ABB RobotStudio station: Proyecto_20210527-053903.rsstn

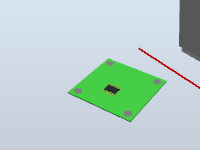
Station Proyecto (saved by RobotStudio 21.1.9443.2)
Controller IRB14000
  mechanical unit ROB_R: IRB14000_0.5_0.5_R, 6 joints, base frame (0, 0, 0) mm
  mechanical unit ROB_R_7: IRB14000_0.5_0.5_R, 1 joints, base frame (0, 0, 0) mm
  mechanical unit ROB_L: IRB14000_0.5_0.5_L, 6 joints, base frame (0, 0, 0) mm
  mechanical unit ROB_L_7: IRB14000_0.5_0.5_L, 1 joints, base frame (0, 0, 0) mm
Layout (positions relative to the parent item):
  - IRB14000_0.5_0.5 [mechanism, from Robots\IRB14000_0.5_0.5__02.rslib] at (0, 0, 0) mm
  - IRB14000_0.5_0.5_R [mechanism, from Robots\IRB14000_0.5_0.5__02.rslib] at (0, 0, 0) mm; joint values [0.0079, -2.3073, -2.3848, 0.4366, 0.2482, 1.2301, -3.4933] (rad or m)
  - IRB14000_0.5_0.5_L [mechanism, from Robots\IRB14000_0.5_0.5__02.rslib] at (0, 0, 0) mm; joint values [-2.0402, -2.3304, 0.9, 0.5715, 0.2248, -0.5734, -1.7213] (rad or m)
  - Part_1 [part] at (100, 0, 0) mm
  - MyTool [mechanism, from Training Objects\myTool.rslib] at (-9.58, -182.61, 198.63) mm, rotated rx -90 ry 76.24 rz -90 deg
  - Chip [part] at (492.85, -76.39, 101.1) mm
  - Drill_holder [mechanism] at (396.94, 21.77, 200.3) mm, rotated rx 106.8 ry 1.53 rz 74.44 deg; joint values [-0.025, 0.0219, 0.0219] (rad or m)
      TCP Tip_holder_mechanism at (-0.08, -53.38, 109.89) mm, rotated rx -73 ry 2 rz -178 deg
      links: L1, L2, L3, L4
  - Part_33 [part]
Attachment: MyTool is attached to IRB14000_0.5_0.5_R / Link7
Attachment: Drill_holder is attached to IRB14000_0.5_0.5_L / Link7
Targets, tools, work objects and paths stored in the station, written as RAPID:
! task T_ROB_R
MODULE CalibData
  PERS tooldata MyTool:=[TRUE,[[31.792631019,0,229.638935148],[0.945518576,0,0.325568154,0]],[1,[0,0,1],[1,0,0,0],0,0,0]];
ENDMODULE

! task T_ROB_R
MODULE Module1
  CONST robtarget Home:=[[177.435607371,-139.377127546,68.621989955],[0.228041545,-0.180578944,0.955893432,-0.040694536],[0,0,-2,4],[-101.964427132,9E+09,9E+09,9E+09,9E+09,9E+09]];
ENDMODULE

! task T_ROB_L
MODULE Module1
  CONST robtarget Home:=[[61.480882858,158.400356438,102.243977191],[0.078264412,0.604906798,-0.79132965,-0.041950353],[0,0,-1,4],[101.964427132,9E+09,9E+09,9E+09,9E+09,9E+09]];
ENDMODULE

! task T_ROB_L
MODULE CalibData
  PERS tooldata Tip_holder_mechanism:=[TRUE,[[-0.077,-53.377,109.892],[0.024406608,0.003647592,0.594886456,-0.803430842]],[0.5,[0,1.6,65.9],[1,0,0,0],0,0,0]];
ENDMODULE

